Fanuc KAREL source: MP0080.KL

-- PROVISIONAL review KL for V940-1; original PC SHA256 ebdfb8ce85e549aceeb47b6b5a3fd5677e3409c06d18a90aa0af9482fcf78705
-- Incomplete behavior may be omitted. Consult companion uncertainty JSON. Do not deploy.
PROGRAM MP0080
%NOLOCKGROUP
-- UNRESOLVED_LOCAL_POOL 8 cells at code offset 65; source declarations unknown
-- DIRECT_LOCAL_WORD_ACCESS alone does not prove INTEGER, REAL, or BOOLEAN
BEGIN
  -- V9_ZERO_TABLE_METADATA_HINT layout=0001; no indexed target words; source/name/runtime held
  -- UNRESOLVED_PC offsets 0-1; opcodes 7B
  -- UNRESOLVED_PC offsets 6-18; opcodes 2D,9D,52,7F
  -- UNRESOLVED_PC offsets 23-28; opcodes 7F,7B
  -- UNRESOLVED_PC offsets 33-49; opcodes 2D,2E,69,7F
  -- UNRESOLVED_PC offsets 54-70; opcodes 7F,2B,2C,7B
  -- UNRESOLVED_PC offsets 75-86; opcodes 2E,23
  -- UNRESOLVED_PC offsets 91-102; opcodes 2E,23
  -- UNRESOLVED_PC offsets 107-118; opcodes 2E,23
  -- UNRESOLVED_PC offsets 123-134; opcodes 2E,23
  -- UNRESOLVED_PC offsets 139-150; opcodes 2E,23
  -- UNRESOLVED_PC offsets 155-166; opcodes 2E,23
  -- UNRESOLVED_PC offsets 171-185; opcodes 2E,22,9D,33,35
  -- UNRESOLVED_PC offsets 190-212; opcodes 22,9D,33,34,21,6B,23
  -- UNRESOLVED_PC offsets 217-221; opcodes 7F
  -- UNRESOLVED_PC offsets 226-242; opcodes 27,27,2E,27,2E,AA
  -- UNRESOLVED_PC offsets 247-251; opcodes 7F
END MP0080
